// Implicitly generated code : DO NOT EDIT
FUNCTION CheckDivDInt : DINT
VAR_INPUT
	divisor:DINT;
END_VAR

// Implicitly generated code : Only an Implementation suggestion
{noflow}
IF divisor = 0 THEN
	CheckDivDInt:=1;
	
	divisionCheckCounter:= divisionCheckCounter + 1;
	
	
ELSE
	CheckDivDInt:=divisor;
END_IF;
{flow}

END_FUNCTION

(* stored: Version 1.1.0.1, ProductVersion 3.1.4024.15
   POU CheckDivDInt: Id {c18cdfdc-3800-408e-852d-c7ac25778675}, SpecialFunc CheckDivInt32 *)
